(*********************************** G.D S.p.A. - Technical Department ***********************************
============= PROGRAM INFO ============
FOLDER:             TBD
MACHINES INVOLVED:  TBD 

============= DESCRIPTION =============
csp machine declaration

============= REVISIONS ===============
Date		Version	 	Author      	Description             
----------	-------		------------  	--------------------------------------------
2019/02/12 	0000.01	 	G.Imbriaco		AccU Change motor with absolute encoder and brake.
										If position_req_mm parameter different from actual_pos_mm and machine reset_edge
										the motor move to position_req then disable again
										Manual movement with basc axis object under test( preset, moving,...)
										All disabled if main accU_Change is not Operational
										
2020/05/11	0000.02		M. Peppo		Added axis_move_condition variable for easy programming accessabilty

**********************************************************************************************************)
(*$R process_ref := prc; $*)
PROGRAM csp_transfer_infeed_accU_depth
VAR
	
	prc:											process;
	prc_path:										STRING;
	
	axis:											axis;
	Slot82_drv:										coe_drive;

	not_in_position:								message;
	axis_restore_absolute_position_fb:				restore_absolute_position_with_retain_fb;

	disable_req:									BOOL:=FALSE;
	position_req_mm:								LREAL:=0.0;(*$P $*)
	move_velocity_req_mms:							LREAL:=10.0;(*$P $*)
	position_req_tolerance_mm:						LREAL:=0.2;	(*$P $*)
	
	axis_status:									axis_status_enum := AXIS_STATUS_PARAMETERS_START;(*$M $*)
	in_position:									BOOL:=FALSE;(*$M $*)	
	actual_position_mm:								LREAL:=0.0; (*$M $*)
	axis_move_condition:							BOOL:=FALSE;
	torque_limit:                                   INT := 5000;    
    torque_limit_old:                               INT;
	
	fsm_status:										csp_transfer_infeed_accU_depth_enum;(*$M $*)
	fsm_next_status:								csp_transfer_infeed_accU_depth_enum;
	fsm_enable_condition:							BOOL:=FALSE;
	debug_state_machine:							BOOL:=FALSE;
	debug_state_machine_one_step:					BOOL:=FALSE;
	NC_encoder_val AT %I*:							DINT;
	
END_VAR
VAR PERSISTENT
	axis_restore_absolute_position_data:			restore_absolute_position_with_retain_struct;
END_VAR

_read_var_input();

_object_manager();

IF NOT objects_running()
THEN
	RETURN;	
END_IF

_read_process_image();

_mode_manager();

CASE process_get_mode(prc) OF
	MODE_ABSENT,
	MODE_INACTIVE:
		RETURN;
	MODE_TEST:
		_handle_process_test();
END_CASE

_set_runtime_properties();

(********************************* BODY *********************************)
//Axis Torque Limit
IF torque_limit <> Torque_limit_old
THEN
    IF coe_drive_write_parameter(
        index:=16#7010 ,
        complete_access:= FALSE ,
        sub_index:= 16#0B,
        data_source:= ADR(torque_limit),
        data_lenght:= SIZEOF(torque_limit),
        CONVERSION_this:=csp_transfer_infeed_accU_depth.axis.coe_drive^ ) = COE_DRIVE_RETURN_VALUE_DONE
	THEN
		torque_limit_old := Torque_limit;
	END_IF
END_IF

//Axis move condition
IF csp_main_accuChange.transfer_infeed_accU_depth_move_req 
THEN
	axis_move_condition := TRUE;
ELSE
	axis_move_condition := FALSE;
END_IF

(*FSM Control*)
fsm_enable_condition := axis_is_ok(FALSE, axis)
						AND
						process_subtree_is_ready(prc)
						AND
						process_get_mode(csp_main_accuChange.prc) = MODE_OPERATIONAL
						AND
						axis_restore_absolute_position_fb.o_position_restored
						AND
						axis_move_condition
						AND
						NOT jog_manager_is_jog_axis_active(SMTR61700_TRANSFER_INFEED_DEPTH, csp_main_jogManager.jog_manager_accuchange)
						AND
						NOT disable_req;	
					
IF	(NOT fsm_enable_condition
	OR
	disable_req)
	AND
	fsm_status <> CSP_TRANSFER_INFEED_ACCU_DEPTH_STATUS_DISABLED
	AND
	fsm_status < CSP_TRANSFER_INFEED_ACCU_DEPTH_STATUS_STOP_REQUEST
THEN
	fsm_status	:=	CSP_TRANSFER_INFEED_ACCU_DEPTH_STATUS_STOP_REQUEST;
END_IF

CASE fsm_status OF
	CSP_TRANSFER_INFEED_ACCU_DEPTH_STATUS_NOT_INITIALIZED:
	
        IF	axis_is_ok(return_when_absent := TRUE, CONVERSION_this := axis)
        THEN
            fsm_next_status := CSP_TRANSFER_INFEED_ACCU_DEPTH_STATUS_DISABLED;
        END_IF

		
	CSP_TRANSFER_INFEED_ACCU_DEPTH_STATUS_DISABLED:
	
		IF	fsm_enable_condition
		THEN
			(* Axis with absolute encoder, no home procedure request *)
			fsm_next_status := CSP_TRANSFER_INFEED_ACCU_DEPTH_STATUS_POSITION_CHECK;
		END_IF;
	
		
	CSP_TRANSFER_INFEED_ACCU_DEPTH_STATUS_POSITION_CHECK:

		(* CHECKS IF AXIS IS IN TOLERANCE *)
		IF 	NOT in_position
			AND machine_is_not_running(csp.mch)  
		THEN
			(* NOT IN TOLERANCE - NEED TO ENABLE AND MOVE *)
			fsm_next_status := CSP_TRANSFER_INFEED_ACCU_DEPTH_STATUS_ENABLE_REQUEST;
		END_IF		
	
		
	CSP_TRANSFER_INFEED_ACCU_DEPTH_STATUS_ENABLE_REQUEST:
	
		axis_enable(axis);
		IF axis_is_standstill(axis)
		THEN
			fsm_next_status	:=	CSP_TRANSFER_INFEED_ACCU_DEPTH_STATUS_ENABLED;
		END_IF	

		
	CSP_TRANSFER_INFEED_ACCU_DEPTH_STATUS_ENABLED:
	
		IF axis_move_condition
		THEN
			fsm_next_status	:= CSP_TRANSFER_INFEED_ACCU_DEPTH_STATUS_CHECK_MOVE;	
		END_IF
		
		
	(* CHECKS TO SEE IF OUTRUN IS NEEDED *)
	CSP_TRANSFER_INFEED_ACCU_DEPTH_STATUS_CHECK_MOVE:
	
		IF position_req_mm >= axis.actual_position
		THEN
			fsm_next_status := CSP_TRANSFER_INFEED_ACCU_DEPTH_STATUS_OUTRUN;
		ELSE
			fsm_next_status := CSP_TRANSFER_INFEED_ACCU_DEPTH_STATUS_ABS_MOVE_REQUEST;
		END_IF
		
	
	CSP_TRANSFER_INFEED_ACCU_DEPTH_STATUS_OUTRUN:
	
		IF	axis_is_standstill(axis)
		THEN
			 axis_move_absolute(
				position 		:= position_req_mm + 2,
				velocity 		:= move_velocity_req_mms,
				direction		:= AXIS_SHORTEST_WAY,
				acceleration 	:= csp_main_accuChange.CONSTANTS.MAX_ACCELERATION_MMpSEC2,
				deceleration 	:= csp_main_accuChange.CONSTANTS.MAX_DECELERATION_MMpSEC2,
				jerk 			:= csp_main_accuChange.CONSTANTS.MAX_JERK_MMpSEC3, 
				buffer_mode 	:= AXIS_BUFFER_MODE_BUFFERED,
				CONVERSION_this := axis
				); 			
		END_IF
		
		IF axis_is_absolute_moving(axis)
		THEN
			fsm_next_status	:=	CSP_TRANSFER_INFEED_ACCU_DEPTH_STATUS_WAIT_FOR_OUTRUN;
		END_IF
		
		
	CSP_TRANSFER_INFEED_ACCU_DEPTH_STATUS_WAIT_FOR_OUTRUN:
	
		IF	axis_is_standstill(axis)
		THEN
			fsm_next_status := CSP_TRANSFER_INFEED_ACCU_DEPTH_STATUS_ABS_MOVE_REQUEST;
		END_IF
	
		
	CSP_TRANSFER_INFEED_ACCU_DEPTH_STATUS_ABS_MOVE_REQUEST:

		IF	axis_is_standstill(axis)
		THEN
			 axis_move_absolute(
				position 		:= position_req_mm,
				velocity 		:= move_velocity_req_mms,
				direction		:= AXIS_SHORTEST_WAY,
				acceleration 	:= csp_main_accuChange.CONSTANTS.MAX_ACCELERATION_MMpSEC2,
				deceleration 	:= csp_main_accuChange.CONSTANTS.MAX_DECELERATION_MMpSEC2,
				jerk 			:= csp_main_accuChange.CONSTANTS.MAX_JERK_MMpSEC3, 
				buffer_mode 	:= AXIS_BUFFER_MODE_BUFFERED,
				CONVERSION_this := axis
				); 			
		END_IF
		
		IF axis_is_absolute_moving(axis)
		THEN
			fsm_next_status	:=	CSP_TRANSFER_INFEED_ACCU_DEPTH_STATUS_ABS_MOVING;
		END_IF

		
	CSP_TRANSFER_INFEED_ACCU_DEPTH_STATUS_ABS_MOVING:

		IF axis_is_standstill(axis)
		THEN
			fsm_next_status := CSP_TRANSFER_INFEED_ACCU_DEPTH_STATUS_DISABLE_REQUEST;
		END_IF
		
		
	CSP_TRANSFER_INFEED_ACCU_DEPTH_STATUS_STOP_REQUEST:

		axis_stop(
		    deceleration 	:= csp_main_accuChange.CONSTANTS.MAX_DECELERATION_MMpSEC2,
		    jerk 			:= csp_main_accuChange.CONSTANTS.MAX_JERK_MMpSEC3,
		    CONVERSION_this 			:= axis);

		IF 	axis_is_standstill(axis)
			OR
			NOT axis_is_ok(FALSE, axis)
			OR
			axis_is_disabled(axis)
		THEN
			fsm_next_status := CSP_TRANSFER_INFEED_ACCU_DEPTH_STATUS_DISABLE_REQUEST;
		END_IF

		
	CSP_TRANSFER_INFEED_ACCU_DEPTH_STATUS_DISABLE_REQUEST:
	
   		axis_disable(axis);
        IF	axis_is_disabled(axis)
        THEN
            fsm_next_status := CSP_TRANSFER_INFEED_ACCU_DEPTH_STATUS_DISABLED;
        END_IF;
END_CASE;

IF NOT debug_state_machine
	OR
	debug_state_machine_one_step
THEN
	fsm_status := fsm_next_status;
	debug_state_machine_one_step := FALSE;
END_IF

(************************************************************************)
_brand_change();

_handle_messages();

_write_output();

ACTION _brand_change:
;
END_ACTION

ACTION _handle_messages:
IF in_position OR csp_main_jogManager.jog_is_active
THEN
	;//process_message_reset(not_in_position);
ELSE
	IF csp_main_accuChange.machine_size_complete = FALSE
	THEN
		;//process_message_reset(not_in_position);
	ELSE
		;//process_message_set(errorID_1:= 1, errorID_2:= 0, errorID_3:= 0, CONVERSION_this:= not_in_position);
	END_IF
END_IF
END_ACTION

ACTION _handle_process_test:
;
END_ACTION

ACTION _mode_manager:
IF process_mode_req_is_pending(prc)
THEN
    process_apply_mode_req_first_step(prc);
    CASE process_get_mode(prc) OF
        MODE_TO_ABSENT:
			;
        MODE_TO_INACTIVE:
			;
        MODE_TO_TEST:
			;
        MODE_TO_OPERATIONAL:
			;
    END_CASE
    process_apply_mode_req_second_step(prc);
END_IF
END_ACTION

ACTION _object_manager:
IF objects_initialization()
THEN
	sub_process_init(
		object_name								:= 'csp_transfer_infeed_accU_depth.prc', 
		process									:= csp_transfer_infeed_accU.prc, 
		CONVERSION_this							:= prc);
		
	prc_path 									:= process_get_path(prc);

	IF csp_main_configurator.Physical_hw 
	THEN
		axis_init(
			object_name							:= CONCAT(prc_path, '_axis'), 
			axis_type							:= AXIS_TYPE_SERVO, 
			encoder_scaling_factor				:= 0.000003719329833, // 22.5171mm_rev
 			modulo								:= 1024, 
  			process								:= prc, 
			CONVERSION_this						:= axis);
			
		axis_init_absolute_encoder_preset(	
			position							:=	200,
			CONVERSION_this						:=	axis);

		axis_add_safety_integrated_series(
			safety_integrated_series			:= csp_transfer_main_safety_accUChange.sis,
			CONVERSION_this						:= axis);
		axis_set_brake_type(AXIS_BRAKE_DRIVE_CMD, axis);
	ELSE
		axis_init(
			object_name 						:= CONCAT(prc_path, '_axis'),
			axis_type 							:= AXIS_TYPE_VIRTUAL,
			encoder_scaling_factor 				:= G_VIRTUAL_ENCODER_SCALING_FACTOR_DEGPINC,
			modulo 								:= G_MODULO_360_DEG,
			process 							:= prc,
			CONVERSION_this 					:= axis);
	END_IF
		
	axis_set_rotation_direction(
		invert_encoder_counting					:= TRUE,
		invert_motor_polarity					:= TRUE,
		CONVERSION_this							:= axis);

	coe_drive_init(
		object_name 							:= CONCAT(prc_path, '_Slot82_drv'),
		device_name 							:= 'IO61600Slot82 (EL7221)',
		vendor 									:= DRIVE_BECKHOFF_EL72x1,
		mode 									:= COE_DRIVE_MODE_DRIVEN_BY_AXIS,
		ethercat_master							:= csp_main.cabinet_transfer_ethercat_master,
		process									:= prc,
		CONVERSION_this 						:= Slot82_drv);

	axis_add_coe_drive(
		coe_drive								:= Slot82_drv,
		CONVERSION_this							:= axis);
	
	axis_set_max_dynamic(
		reference_velocity						:=	csp_main_accuChange.CONSTANTS.MAX_VELOCITY_MMpSEC,
		velocity								:=	csp_main_accuChange.CONSTANTS.MAX_VELOCITY_MMpSEC,
		acceleration							:=	csp_main_accuChange.CONSTANTS.MAX_ACCELERATION_MMpSEC2,
		deceleration							:=	csp_main_accuChange.CONSTANTS.MAX_DECELERATION_MMpSEC2,
		jerk									:=	csp_main_accuChange.CONSTANTS.MAX_JERK_MMpSEC3,
		following_error							:=	csp_main_accuChange.CONSTANTS.MAX_FOLLOWING_ERROR_MM,
		CONVERSION_this							:=	axis);
	
	jog_manager_add_axis(
		list_index								:= SMTR61700_TRANSFER_INFEED_DEPTH,
		axis									:= axis,
		master_axis								:= FALSE,
		jog_type								:= JOG_TYPE_LINEAR,
		sw_limit_positive						:= 200,
		sw_limit_negative						:= 0,
		CONVERSION_this							:= csp_main_jogManager.jog_manager_accuchange);
		

	process_message_init(
		object_name:= CONCAT(prc_path, '_not_in_position'), 
		behaviour:= MESSAGE_BEHAVIOUR_STATE, 
		reset_timeout:= 0, 
		disableable:= TRUE, 
		individual_reset:= FALSE, 
		machine_reaction:= MACHINE_REACTION_STOP_IN_PHASE_ONE, 
		typology:= MESSAGE_TYPOLOGY_ABNORMAL, 
		process:= prc, 
		CONVERSION_this:= not_in_position);
		
END_IF

IF objects_running()
THEN
	process_cycle(prc);
	axis_cycle(axis);
	coe_drive_cycle(Slot82_drv); 
END_IF
END_ACTION

ACTION _read_process_image:
axis_restore_absolute_position_fb(
	io_retain_data				:= axis_restore_absolute_position_data, 
	io_axis						:= axis);
END_ACTION

ACTION _read_var_input:
;
END_ACTION

ACTION _set_runtime_properties:

axis_status := axis_get_status(axis);
actual_position_mm :=axis_get_actual_incremental_position(axis); (* axis_get_actual_modulo_position(axis); only with modulo*)

IF ABS(position_req_mm - actual_position_mm)< position_req_tolerance_mm
	OR
	process_get_mode(prc)= MODE_ABSENT
	OR
	process_get_mode(csp_main_accuChange.prc) = MODE_ABSENT
THEN
	in_position := TRUE;
ELSE
	in_position := FALSE; 	
END_IF
END_ACTION

ACTION _write_output:
;
END_ACTION

END_PROGRAM

(* stored: Version 1.1.0.1, ProductVersion 3.1.4024.3
   POU csp_transfer_infeed_accU_depth: Id {ced3a087-1219-4ade-bf6f-6ccb8a17dd0c}, SpecialFunc None
   Action _brand_change: Id {64bb9a48-f0aa-4eaf-b88d-ebb4d908887c}
   Action _handle_messages: Id {6e4fc461-b33e-4dfd-8835-8c3985705e76}
   Action _handle_process_test: Id {80ee279e-1e8a-4223-ac12-dea6a914064e}
   Action _mode_manager: Id {be63499a-285c-4b6e-b85d-89ed9802575c}
   Action _object_manager: Id {9844e982-b788-4b8f-b1a1-3dfea3085d19}
   Action _read_process_image: Id {9b973d6d-b95f-49bb-8850-629ca4861bf7}
   Action _read_var_input: Id {e1576158-b639-4fe1-9f9f-ec39f9261d4a}
   Action _set_runtime_properties: Id {7ea5d6ae-fbb6-4a7b-9a74-62b1148bc19e}
   Action _write_output: Id {f39953c2-e2e4-4561-82e2-ce4ecf3e896f} *)
